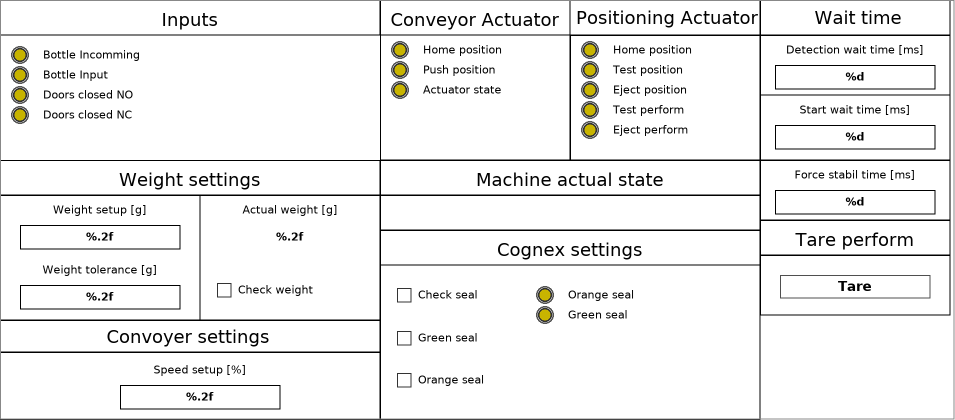
VISUALIZATION vDetectionTunelFrame  // 955x420
VAR_IN_OUT
	stInOuts : stDetectionTunelInOuts;
	stParams : stDetectionTunelParams;
	iWorkStep	: INT;
END_VAR
    Rectangle (760,220 190x35)
    Rectangle (760,0 190x35)
    Rectangle (0,352 380x68)
    Rectangle (380,160 380x35)
    Rectangle (0,195 200x125)
    Rectangle (380,230 380x190)
    Rectangle (0,195 380x125)
    Rectangle (380,0 380x35)
    Lamp1 (10,45 20x20), variable: stInOuts.bBottleIncomming, style: Lamp-Lamp1-Yellow
    Lamp1 (10,65 20x20), variable: stInOuts.bBottleInput, style: Lamp-Lamp1-Yellow
    Lamp1 (10,85 20x20), variable: stInOuts.bDorsClosedNO, style: Lamp-Lamp1-Yellow
    Lamp1 (10,105 20x20), variable: stInOuts.bDorsClosedNC, style: Lamp-Lamp1-Yellow
    Label (40,45 150x20), "Bottle Incomming"
    Label (40,65 150x20), "Bottle Input"
    Label (40,85 150x20), "Doors closed NO"
    Label (40,105 150x20), "Doors closed NC"
    Rectangle (0,0 380x35)
    Label (0,5 380x30), "Inputs"
    Rectangle (380,0 190x160)
    Rectangle (570,35 190x125)
    Label (380,5 190x30), "Conveyor Actuator"
    Rectangle (0,160 380x35)
    Label (420,40 150x20), "Home position"
    Lamp1 (390,40 20x20), variable: stInOuts.bActuatorConvoyerHome, style: Lamp-Lamp1-Yellow
    Lamp1 (390,60 20x20), variable: stInOuts.bActuatorConvoyerPush, style: Lamp-Lamp1-Yellow
    Lamp1 (390,80 20x20), variable: stInOuts.bActuatorConvoyerPush, style: Lamp-Lamp1-Yellow
    Label (420,60 150x20), "Push position"
    Label (420,80 150x20), "Actuator state"
    Label (380,165 380x30), "Machine actual state"
    Rectangle (380,195 380x35), text list: 'tlDetectionTunel', text index: iWorkStep
    Label (0,165 380x30), "Weight settings"
    Rectangle (20,225 160x24), "%.2f", text variable: stParams.rBottleLoad, input disabled if: NOT GVL.fbUserLogin.bPermissionGranted
        OnMouseClick: write the text variable via Default, min 100, max 1000, format %d
    Label (10,200 180x20), "Weight setup [g]"
    Label (572,3 190x30), "Positioning Actuator"
    Label (610,40 150x20), "Home position"
    Label (610,60 150x20), "Test position"
    Label (610,80 150x20), "Eject position"
    Label (610,100 150x20), "Test perform"
    Lamp1 (580,40 20x20), variable: stInOuts.bActuatorHome, style: Lamp-Lamp1-Yellow
    Lamp1 (580,60 20x20), variable: stInOuts.bActuatorTestLoad, style: Lamp-Lamp1-Yellow
    Lamp1 (580,80 20x20), variable: stInOuts.bActuatorPush, style: Lamp-Lamp1-Yellow
    Lamp1 (580,100 20x20), variable: stInOuts.bActuatorPositioning, style: Lamp-Lamp1-Yellow
    Label (610,120 150x20), "Eject perform"
    Lamp1 (580,120 20x20), variable: stInOuts.bActuatorDropBottle, style: Lamp-Lamp1-Yellow
    Label (10,260 180x20), "Weight tolerance [g]"
    Rectangle (20,285 160x24), "%.2f", text variable: stParams.rBottleLoadTolerance, input disabled if: NOT GVL.fbUserLogin.bPermissionGranted
        OnMouseClick: write the text variable via Default, min 1, max 40, format %d
    Rectangle (210,225 160x24), "%.2f", text variable: stInOuts.rLoadCell
    Label (200,200 180x20), "Actual weight [g]"
    Rectangle (380,230 380x35)
    Label (380,235 380x30), "Cognex settings"
    Checkbox (215,275 150x30), "Check weight", variable: stParams.bWeightCheck, input disabled if: NOT GVL.fbUserLogin.bPermissionGranted
    Checkbox (395,280 150x30), "Check seal", variable: stParams.bCognexEnable, input disabled if: NOT GVL.fbUserLogin.bPermissionGranted
    Lamp1 (535,285 20x20), variable: stInOuts.stCognex.bIn1, style: Lamp-Lamp1-Yellow
    Label (565,285 150x20), "Orange seal"
    Label (565,305 150x20), "Green seal"
    Lamp1 (535,305 20x20), variable: stInOuts.stCognex.bInOut2, style: Lamp-Lamp1-Yellow
    Label (-2,322 380x30), "Convoyer settings"
    Label (110,360 180x20), "Speed setup [%]"
    Rectangle (120,385 160x24), "%.2f", text variable: stParams.rConvoyerSpeed, input disabled if: NOT GVL.fbUserLogin.bPermissionGranted
        OnMouseClick: write the text variable via Default, format %d
    Rectangle (0,320 380x32)
    Checkbox (395,323 150x30), "Green seal", variable: stParams.bGreenExpected, input disabled if: NOT GVL.fbUserLogin.bPermissionGranted
    Checkbox (395,365 150x30), "Orange seal", variable: stParams.bOrangeExpected, input disabled if: NOT GVL.fbUserLogin.bPermissionGranted
    Rectangle (760,35 190x125)
    Label (763,3 190x30), "Wait time"
    Rectangle (760,35 190x60)
    Label (760,35 190x30), "Detection wait time [ms]"
    Label (760,95 190x30), "Start wait time [ms]"
    Rectangle (760,160 190x60)
    Label (760,160 190x30), "Force stabil time [ms]"
    Rectangle (775,190 160x24), "%d", text variable: stParams.iForceStabilTime, input disabled if: NOT GVL.fbUserLogin.bPermissionGranted
        OnMouseClick: write the text variable via Default, format %d
    Rectangle (775,125 160x24), "%d", text variable: stParams.iStartWaitTime, input disabled if: NOT GVL.fbUserLogin.bPermissionGranted
        OnMouseClick: write the text variable via Default, format %d
    Rectangle (775,65 160x24), "%d", text variable: stParams.iDetectionWaitTime, input disabled if: NOT GVL.fbUserLogin.bPermissionGranted
        OnMouseClick: write the text variable via Default, format %d
    Label (760,225 190x30), "Tare perform"
    Rectangle (760,255 190x60)
    Rectangle (780,275 150x23), "Tare", input disabled if: NOT GVL.fbUserLogin.bPermissionGranted
        OnMouseClick: toggle stInOuts.bTarePerform
END_VISUALIZATION

(* stored: Version 1.1.0.1, ProductVersion 3.1.4024.13
   Visu vDetectionTunelFrame: Id {690f2621-797d-4627-8729-61487e2cda88} *)
